(* CoDeSys 2.3.9.41 project: warm.pro *)
(* Libraries: STANDARD.LIB 4.10.05 10:14:46, IECSFC.LIB 13.4.06 14:51:28, SYSLIBTIME.LIB 20.2.06 13:31:16, SYSTASKINFO.LIB 20.2.06 13:31:38, ANALYZATION.LIB 5.10.99 08:05:06, SYSLIBCALLBACK.LIB 20.2.06 13:31:08 *)

(* PLC configuration (modules and I/O channels)
Discrete input 6 bit [ID100] node 0, in %IB0 out %QB0 {Filtrationtime = 10; Filtrationtime = 10; Filtrationtime = 10; Filtrationtime = 10; Filtrationtime = 10; Filtrationtime = 10; Visibility = No; PinCount = 6; WatchDogPeriod = 1000; PollPeriod = 1}
  AT %IX0.0 [BitInput]
  AT %IX0.1 [BitInput]
  AT %IX0.2 [BitInput]
  AT %IX0.3 [BitInput]
  AT %IX0.4 [BitInput]
  AT %IX0.5 [BitInput]
Discrete output 4 bit [ID101] node 1, in %IB1 out %QB1 {PinCount = 4; SafeValueBool = FALSE; SafeValueBool = FALSE; SafeValueBool = FALSE; SafeValueBool = FALSE; Visibility = No}
  AT %QX1.0 [BitOutput]
  AT %QX1.1 [BitOutput]
  AT %QX1.2 [BitOutput]
  AT %QX1.3 [BitOutput]
Special output [ID104] node 2, in %IB2 out %QB2 {Visibility = No; PinCount = 1}
  AT %QX2.0 [BitOutput] Special output
AI0_presIN AT %ID3.0 [FloatInput] Value
AT %IW3.1 [WordInput] Circular time
Analog Input [ID107] node 0, in %IB3.0 out %QB3.0
AI1_presOUT AT %ID4.0 [FloatInput] Value
AT %IW4.1 [WordInput] Circular time
Analog Input [ID107] node 0, in %IB4.0 out %QB4.0
Unifed signal sensor [ID700] node 5, in %IB5 out %QB5 {Type_of_sensor700 = IT_0_20; measure_interval = 0.5; ainlow = 0; ainhigh = 20; first_cor_point = 0; first_delta = 0; second_cor_point = 0; second_delta = 0; third_cor_point = 0; third_delta = 0; Visibility = No}
  AI2_outsideTemp AT %ID5.0 [FloatInput] Value
  AT %IW5.1 [WordInput] Circular time
  Analog Input [ID107] node 0, in %IB5.0 out %QB5.0
Unifed signal sensor [ID700] node 6, in %IB6 out %QB6 {Type_of_sensor700 = IT_0_20; measure_interval = 0.5; ainlow = 0; ainhigh = 20; first_cor_point = 0; first_delta = 0; second_cor_point = 0; second_delta = 0; third_cor_point = 0; third_delta = 0; Visibility = No}
  AT %ID6.0 [FloatInput] Value
  AT %IW6.1 [WordInput] Circular time
  Analog Input [ID107] node 0, in %IB6.0 out %QB6.0
Analog output [ID106] node 7, in %IB7 out %QB7 {DAC_Type = Voltage 0-10 B; Analog_offset_correction = 0; Analog_full_range_correction = 0; SafeValueFloat = 0; Visibility = No}
  AT %QD7.0 [FloatOutput] Value
Analog output [ID106] node 8, in %IB8 out %QB8 {DAC_Type = Voltage 0-10 B; Analog_offset_correction = 0; Analog_full_range_correction = 0; SafeValueFloat = 0; Visibility = No}
  AT %QD8.0 [FloatOutput] Value
ModBus (Master) [MODBUS_MASTER_ID450] node 9, in %IB9 out %QB9 {Visibility = No}
  AT %QD9.0 [DWordOutput] Last address
  AT %QW9.1 [WordOutput] Last error
  RS-485-1 [COM1_USART] node 0, in %IB9.0 out %QB9.0 {CommunicationSpeed = 11520; Parity = NO PARITY CHECK; BitLength = 8 bits; StopLength = Two stop bits; InterfaceType = RS485; FrameOriented = RTU; Timeout = 0; Visibility = No}
  Universal Modbus device [ID2000] node 1, in %IB9.1 out %QB9.1 {ModuleIP = 10:0:0:223; ServiceTimeout = 150; TCPport = 502; NetMode = Serial; ModuleSlaveAddress = 3; RequestType = By poll time; PeriodOfService = 3000; Visibility = No; RepeatCounter = 0; ByteSequence = Native}
    AT %QB9.1.0 [ComChannel] Command (0xff - Start)
trm1_temperature AT %IW9.1.0.0 [WordInput]
trm1_setpoint AT %IW9.1.1.0 [WordInput]
trm1_state AT %IW9.1.2.0 [WordInput]
trm1_writeSetpoint AT %QW9.1.3.0 [WordOutput]
Universal Modbus device [ID2000] node 2, in %IB9.2 out %QB9.2 {ModuleIP = 10:0:0:223; ServiceTimeout = 150; TCPport = 502; NetMode = Serial; ModuleSlaveAddress = 4; RequestType = By poll time; PeriodOfService = 3000; Visibility = No; RepeatCounter = 0; ByteSequence = Native}
  AT %QB9.2.0 [ComChannel] Command (0xff - Start)
trm1_temperature AT %IW9.2.0.0 [WordInput]
trm1_setpoint AT %IW9.2.1.0 [WordInput]
trm1_state AT %IW9.2.2.0 [WordInput]
trm1_writeSetpoint AT %QW9.2.3.0 [WordOutput]
Universal Modbus device [ID2000] node 3, in %IB9.3 out %QB9.3 {ModuleIP = 10:0:0:223; ServiceTimeout = 150; TCPport = 502; NetMode = Serial; ModuleSlaveAddress = 5; RequestType = By poll time; PeriodOfService = 2000; Visibility = No; RepeatCounter = 0; ByteSequence = Trace_mode}
  AT %QB9.3.0 [ComChannel] Command (0xff - Start)
fc_frequency AT %IW9.3.0.0 [WordInput]
fc_setpoint AT %ID9.3.1.0 [DWordInput]
fc_power AT %ID9.3.2.0 [DWordInput]
fc_currency AT %ID9.3.3.0 [DWordInput]
fc_pressure AT %ID9.3.4.0 [DWordInput]
fc_writeSetpoint AT %QD9.3.5.0 [DWordOutput]
Modbus [MODBUS_ID302] node 0, in %IB10.0 out %QB10.0
  Debug RS-232 [DEBUG_USART] node 0, in %IB10.0.0 out %QB10.0.0 {CommunicationSpeed = 11520; Parity = EVEN; BitLength = 8 bits; StopLength = One stop bit; InterfaceType = RS232; FrameOriented = RTU; Timeout = 0; Visibility = No}
8 bits [8Bit] node 1, in %IB10.1 out %QB10.1
  AT %QB10.1.0 [ByteOutput]
8 bits [8Bit] node 2, in %IB10.2 out %QB10.2
  AT %QB10.2.0 [ByteOutput]
  AT %QB10.3.0 [ByteOutput]
  pan_weekDays AT %QB10.4.0 [ByteOutput]
  pan_holyDays AT %QB10.5.0 [ByteOutput]
pan_trm1_temp AT %QW10.6.0 [WordOutput]
pan_trm1_set AT %QW10.7.0 [WordOutput]
pan_trm2_temp AT %QW10.8.0 [WordOutput]
pan_trm2_set AT %QW10.9.0 [WordOutput]
pan_fc_freq AT %QW10.10.0 [WordOutput]
pan_fc_freq AT %QW10.11.0 [WordOutput]
pan_fc_pow AT %QW10.12.0 [WordOutput]
pan_fc_pres AT %QW10.13.0 [WordOutput]
pan_fc_set AT %QW10.14.0 [WordOutput]
pan_presIN_4ma AT %QW10.15.0 [WordOutput]
pan_presIN_20ma AT %QW10.16.0 [WordOutput]
pan_presOUT_4ma AT %QW10.17.0 [WordOutput]
pan_presOUT_20ma AT %QW10.18.0 [WordOutput]
pan_weekday_set AT %QW10.19.0 [WordOutput]
pan_holyday_set AT %QW10.20.0 [WordOutput]
pan_weekday_onHH AT %QW10.21.0 [WordOutput]
pan_weekday_onMM AT %QW10.22.0 [WordOutput]
pan_holyday_onHH AT %QW10.23.0 [WordOutput]
pan_holyday_onMM AT %QW10.24.0 [WordOutput]
pan_weekday_offHH AT %QW10.25.0 [WordOutput]
pan_weekday_offMM AT %QW10.26.0 [WordOutput]
pan_holyday_offHH AT %QW10.27.0 [WordOutput]
pan_holyday_offMM AT %QW10.28.0 [WordOutput]
pan_soldierTime AT %QW10.29.0 [WordOutput]
*)

(* Global variable list: Global_Variables *)
VAR_GLOBAL
(* Times *)
	GetTime: CurTimeEx;
	TimeAndDate: SystemTimeDate;
	Sys_Time: SysTime64;
END_VAR

(* POU PLC_PRG, ST *)
PROGRAM PLC_PRG
VAR


	trmGvs_setpoint, trmHeat_setpoint : WORD;
	fc_setpoint : WORD;

	presIN, presIN_4ma, presIN_20ma : WORD;
	presOUT, presOUT_4ma, presOUT_20ma : WORD;

	weekday_setpoint, holyday_setpoint : WORD;
	weekday_byTime, holyday_byTime : BOOL;
	weekday_onHH, holyday_onHH : WORD;
	weekday_onMM, holyday_onMM : WORD;
	weekday_offHH, holyday_offHH : WORD;
	weekday_offMM, holyday_offMM : WORD;

	weekDays, holyDays : WORD;

	HeatStart, HeatStarted : BOOL;
	outsideTemp, nowHoly : WORD;
	timeToHeatWeek, timeToHeatHoly : BOOL;

	soldierTime : TIME;
	soldierTimer : TON;
	soldierOver : BOOL;
	fc_start : BOOL;

	(* heating mode *)
	airLow, trmLow : WORD;
	airHigh, trmHigh : WORD;

END_VAR
VAR RETAIN
	save_trmGvs_setpoint, save_trmHeat_setpoint : WORD;
	save_fc_setpoint : WORD;

	save_presIN, save_presIN_4ma, save_presIN_20ma : WORD;
	save_presOUT, save_presOUT_4ma, save_presOUT_20ma : WORD;

	save_weekday_setpoint, save_holyday_setpoint : WORD;
	save_weekday_byTime, save_holyday_byTime : BOOL;
	save_weekday_onHH, save_holyday_onHH : WORD;
	save_weekday_onMM, save_holyday_onMM : WORD;
	save_weekday_offHH, save_holyday_offHH : WORD;
	save_weekday_offMM, save_holyday_offMM : WORD;

	save_weekDays, save_holyDays : WORD;

	save_soldierTime : TIME;
END_VAR
Calibration;
END_PROGRAM
ACTION Calibration:
presIN := presIN_4ma  + ( REAL_TO_INT( AI0_presIN * 100 ) - 400 ) * ( presIN_20ma - presIN_4ma ) / 1600; (* wordpres := .... точность 0.01 *)

IF AI0_presIN < 4.0 THEN
	presIN := 0;
END_IF;

presOUT := presOUT_4ma  + ( REAL_TO_INT( AI1_presOUT * 100 ) - 400 ) * ( presOUT_20ma - presOUT_4ma ) / 1600; (* wordpres := .... точность 0.01 *)

IF AI1_presOUT < 4.0 THEN
	presOUT := 0;
END_IF;
END_ACTION
ACTION DetermineHoly:
CASE TimeAndDate.DayOfWeek OF
	1 : IF hMON
	     	THEN nowHoly := TRUE;
		ELSE nowHoly := FALSE;
	     END_IF;

	2 : IF hTUE
	     	THEN nowHoly := TRUE;
		ELSE nowHoly := FALSE;
	     END_IF;

      3 : IF hWED
	     	THEN nowHoly := TRUE;
		ELSE nowHoly := FALSE;
	     END_IF;

      4 : IF hTHU
	     	THEN nowHoly := TRUE;
		ELSE nowHoly := FALSE;
	     END_IF;

      5 : IF hFRI
	     	THEN nowHoly := TRUE;
		ELSE nowHoly := FALSE;
	     END_IF;

      6 : IF hSAT
	     	THEN nowHoly := TRUE;
		ELSE nowHoly := FALSE;
	     END_IF;

      0 : IF hSUN
	     	THEN nowHoly := TRUE;
		ELSE nowHoly := FALSE;
	     END_IF;
END_CASE;
END_ACTION
ACTION Heating:
(* проверка условий запуска *)

IF nowHoly THEN
	IF ( holyday_onHH = TimeAndDate.Hour ) AND ( holyday_onMM = TimeAndDate.Minute ) AND ( TimeAndDate.Second = 0 )
		THEN timeToHeatHoly := TRUE;
	END_IF;

	IF ( holyday_offHH = TimeAndDate.Hour ) AND ( holyday_offMM = TimeAndDate.Minute ) AND ( TimeAndDate.Second = 0 )
		THEN timeToHeatHoly := FALSE;
	END_IF;
ELSE
	IF ( weekday_onHH = TimeAndDate.Hour ) AND ( weekday_onMM = TimeAndDate.Minute ) AND ( TimeAndDate.Second = 0 )
		THEN timeToHeatWeek := TRUE;
	END_IF;

	IF ( weekday_offHH = TimeAndDate.Hour ) AND ( weekday_offMM = TimeAndDate.Minute ) AND ( TimeAndDate.Second = 0 )
		THEN timeToHeatWeek := FALSE;
	END_IF;
END_IF;


IF nowHoly THEN
	IF holyday_byTime THEN
		IF ( outsideTemp < holyday_setpoint ) AND  timeToHeatHoly THEN
			HeatStart := TRUE;
		ELSE
			HeatStart := FALSE;
		END_IF;
	ELSE
		IF outsideTemp < holyday_setpoint THEN
			HeatStart := TRUE;
		ELSE
			HeatStart := FALSE;
		END_IF;
	END_IF;
ELSE
	IF weekday_byTime THEN
		IF ( outsideTemp < weekday_setpoint ) AND  timeToHeatWeek THEN
			HeatStart := TRUE;
		ELSE
			HeatStart := FALSE;
		END_IF;
	ELSE
		IF outsideTemp < weekday_setpoint THEN
			HeatStart := TRUE;
		ELSE
			HeatStart := FALSE;
		END_IF;
	END_IF;
END_IF;


(* пуск системы отопления *)
soldierTimer(IN:= HeatStart, PT:=soldierTime, Q=>soldierOver, ET=> );

IF HeatStart AND NOT HeatStarted THEN
	fc_start := TRUE;
	IF soldierOver THEN

	END_IF;
END_IF;

(* останов системы отопления *)
IF NOT HeatStart AND HeatStarted THEN
	fc_start := FALSE;

END_IF;
END_ACTION
ACTION Holydays:
IF wMON = hMON THEN
	wMON := NOT hMON;
END_IF;

IF wTUE = hTUE THEN
	wTUE := NOT hTUE;
END_IF;

IF wWED = hWED THEN
	wWED := NOT hWED;
END_IF;

IF wTHU = hTHU THEN
	wTHU := NOT hTHU;
END_IF;

IF wFRI = hFRI THEN
	wFRI := NOT hFRI;
END_IF;

IF wSAT = hSAT THEN
	wSAT := NOT hSAT;
END_IF;

IF wSUN = hSUN THEN
	hSUN := NOT wSUN;
END_IF;
END_ACTION
ACTION Input:
IF pan_trm1_set <> trmGvs_setpoint THEN
	save_trmGvs_setpoint := pan_trm1_set;
	trmGvs_setpoint := pan_trm1_set;
END_IF;

IF pan_trm2_set <> trmHeat_setpoint THEN
	save_trmHeat_setpoint := pan_trm2_set;
	trmHeat_setpoint := pan_trm2_set;
END_IF;

IF pan_fc_set <> fc_setpoint THEN
	save_fc_setpoint := pan_fc_set;
	fc_setpoint := pan_fc_set;
END_IF;

IF pan_presIN_4ma <> presIN_4ma THEN
	save_presIN_4ma := pan_presIN_4ma;
	presIN_4ma := pan_presIN_4ma;
END_IF;

IF pan_presIN_20ma <> presIN_20ma THEN
	save_presIN_20ma := pan_presIN_20ma;
	presIN_20ma := pan_presIN_20ma;
END_IF;

IF pan_presOUT_4ma <> presOUT_4ma THEN
	save_presOUT_4ma := pan_presOUT_4ma;
	presOUT_4ma := pan_presOUT_4ma;
END_IF;

IF pan_presOUT_20ma <> presOUT_20ma THEN
	save_presOUT_20ma := pan_presOUT_20ma;
	presOUT_20ma := pan_presOUT_20ma;
END_IF;

IF pan_weekday_set <> weekday_setpoint THEN
	save_weekday_setpoint := pan_weekday_set;
	weekday_setpoint := pan_weekday_set;
END_IF;

IF pan_holyday_set <> holyday_setpoint THEN
	save_holyday_setpoint := pan_holyday_set;
	holyday_setpoint := pan_holyday_set;
END_IF;

IF pan_weekday_byTime <> weekday_byTime THEN
	save_weekday_byTime := pan_weekday_byTime;
	weekday_byTime := pan_weekday_byTime;
END_IF;

IF pan_holyday_byTime <> holyday_byTime THEN
	save_holyday_byTime := pan_holyday_byTime;
	holyday_byTime := pan_holyday_byTime;
END_IF;

IF pan_weekday_onHH <> weekday_onHH THEN
	save_weekday_onHH := pan_weekday_onHH;
	weekday_onHH := pan_weekday_onHH;
END_IF;

IF pan_weekday_onMM <> weekday_onMM THEN
	save_weekday_onMM := pan_weekday_onMM;
	weekday_onMM := pan_weekday_onMM;
END_IF;

IF pan_holyday_onHH <> holyday_onHH THEN
	save_holyday_onHH := pan_holyday_onHH;
	holyday_onHH := pan_holyday_onHH;
END_IF;

IF pan_holyday_onMM <> holyday_onMM THEN
	save_holyday_onMM := pan_holyday_onMM;
	holyday_onMM := pan_holyday_onMM;
END_IF;


IF pan_weekday_offHH <> weekday_offHH THEN
	save_weekday_offHH := pan_weekday_offHH;
	weekday_offHH := pan_weekday_offHH;
END_IF;

IF pan_weekday_offMM <> weekday_offMM THEN
	save_weekday_offMM := pan_weekday_offMM;
	weekday_offMM := pan_weekday_offMM;
END_IF;

IF pan_holyday_offHH <> holyday_offHH THEN
	save_holyday_offHH := pan_holyday_offHH;
	holyday_offHH := pan_holyday_offHH;
END_IF;

IF pan_holyday_offMM <> holyday_offMM THEN
	save_holyday_offMM := pan_holyday_offMM;
	holyday_offMM := pan_holyday_offMM;
END_IF;

IF BYTE_TO_WORD ( pan_weekDays ) <> weekDays THEN
	save_weekDays := BYTE_TO_WORD ( pan_weekDays );
	weekDays := BYTE_TO_WORD ( pan_weekDays );
	Weekdays;
END_IF;

IF BYTE_TO_WORD ( pan_holyDays ) <> holyDays THEN
	save_holyDays := BYTE_TO_WORD ( pan_holyDays );
	holyDays := BYTE_TO_WORD ( pan_holyDays );
	Holydays;
END_IF;

IF pan_soldierTime <> soldierTime THEN
	save_soldierTime := pan_soldierTime;
	soldierTime := pan_soldierTime;
END_IF;
END_ACTION
ACTION TempMode:

END_ACTION
ACTION Times:
TimeAndDate.Day :=0;
TimeAndDate.DayOfWeek :=0;
TimeAndDate.dwHighMsec :=0;
TimeAndDate.dwLowMSecs :=0;
TimeAndDate.Milliseconds :=0;
TimeAndDate.Minute :=0;
TimeAndDate.Second :=0;
TimeAndDate.Hour :=0;
TimeAndDate.Year :=0;
TimeAndDate.Month :=0;
Sys_time.ulHigh :=0;
Sys_time.ulLow :=0;
GetTime (SystemTime:=Sys_Time , TimeDate:= TimeAndDate);

(*

IF pan_DISTBITS.0 THEN
	TimeAndDate.Minute:=pan_setMMin;
	TimeAndDate.Second:=10;
	TimeAndDate.Hour:=pan_setHH;
	TimeAndDate.Day:=pan_setDD;
	TimeAndDate.Month:=pan_setMM;
	TimeAndDate.Year:=pan_setYYYY;
	GetTime (SystemTime:=Sys_Time , TimeDate:= TimeAndDate);

	pan_DISTBITS.0 := FALSE;
END_IF;

*)
END_ACTION
ACTION Weekdays:
IF wMON = hMON THEN
	hMON := NOT wMON;
END_IF;

IF wTUE = hTUE THEN
	hTUE := NOT wTUE;
END_IF;

IF wWED = hWED THEN
	hWED := NOT wWED;
END_IF;

IF wTHU = hTHU THEN
	hTHU := NOT wTHU;
END_IF;

IF wFRI = hFRI THEN
	hFRI := NOT wFRI;
END_IF;

IF wSAT = hSAT THEN
	hSAT := NOT wSAT;
END_IF;

IF wSUN = hSUN THEN
	hSUN := NOT wSUN;
END_IF;
END_ACTION
